(* CODESYS project 1.project

Project tree, tasks and I/O mapping:
  Device : CODESYS Control Win V3, 3S - Smart Software Solutions GmbH, order no. 305021, version 3.5.11.30
    application Application
      libraries: Standard, * (System)
      task MainTask (cyclic, interval t#20ms, priority 1) calls PLC_PRG
      program PLC_PRG [LD]
*)

// Device/Application/PLC_PRG
PROGRAM PLC_PRG
VAR
	B1: BOOL; //BOTOERIRA
	B2: BOOL; //BOTOERIRA
	S2: BOOL; //SENSOR CORTINA
	S1: BOOL; //SENSOR DE PEÇA
	S4: BOOL; // SENSOR DE INICIO
	K1: BOOL; // CONTATOR 1
	L1: BOOL; // LAMPADA
	M1: BOOL; // MOTOR DE DESCIDA
	S3: BOOL; // SENSOR FIM 
	K2: BOOL; // CONTATRO 2
	M2: BOOL; // VOLTA DO MOTOR
	BE: BOOL; // BOTÃO DE EMERGENCIA
	L2: BOOL; // LAMPADA DE EMERGECIA 
	AUX1: BOOL; //VARIAVEL AXUXILIAR PARA A SITUÇÃO DE B1 OU B2 DESACIONADOS
END_VAR
VAR // added by the converter: edge detectors and wires of the graphical bodies
    _w1, _w2, _w3 : BOOL;
END_VAR

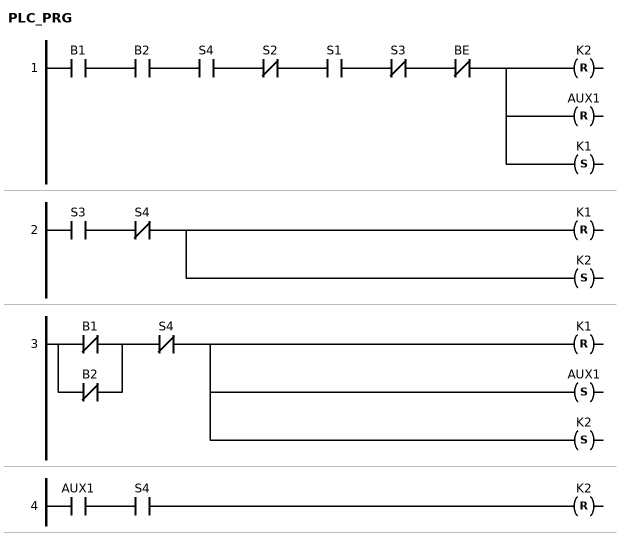
// NETWORK 1
_w1 := B1 AND B2 AND S4 AND NOT S2 AND S1 AND NOT S3 AND NOT BE;
K2 R= _w1;
AUX1 R= _w1;
K1 S= _w1;

// NETWORK 2
_w2 := S3 AND NOT S4;
K1 R= _w2;
K2 S= _w2;

// NETWORK 3
_w3 := (NOT B1 OR NOT B2) AND NOT S4;
K1 R= _w3;
AUX1 S= _w3;
K2 S= _w3;

// NETWORK 4
K2 R= AUX1 AND S4;

END_PROGRAM
